# EPICS autosave request: GALILMUL/iocBoot/iocGALILMUL-IOC-02/GALIL_02_positions.req
file "GALIL_controller_positions.req" P=$(P),CCP=$(CCP)
